(* IEC 61131-3 sources: automationbase/src/OperatingModes, 3 files *)

(* ---- OperatingModes.st ---- *)
NAMESPACE Simatic.Ax.AutomationBase
    /// Operating modes for equipment
    /// Commissioning: Initial setup and testing
    /// Manual: Manual operation with operator control
    /// Automatic: Fully automatic operation with auto-startup
    TYPE
        OperatingModes : (Commissioning, Manual, Automatic) := Manual;
    END_TYPE

END_NAMESPACE

(* ---- IOperatingMode.st ---- *)
NAMESPACE Simatic.Ax.AutomationBase

    {axcode:docs-v0:@simatic-ax/automationbase:OperatingModes.md}
    /// Interface for operating mode providers
    /// Implement this to provide the current operating mode to equipment
    INTERFACE IOperatingMode
        /// Returns the current operating mode (Commissioning, Manual, or Automatic)
        METHOD GetOperatingMode : OperatingModes
        END_METHOD
    END_INTERFACE

END_NAMESPACE

(* ---- OperatingModeManager.st ---- *)
NAMESPACE Simatic.Ax.AutomationBase

    {axcode:docs-v0:@simatic-ax/automationbase:OperatingModes.md}
    /// Generic operating mode manager class
    /// Provides a simple implementation of IOperatingMode with settable mode
    CLASS OperatingModeManager IMPLEMENTS IOperatingMode
        VAR PROTECTED
            /// Current operating mode (default: Manual)
            _currentMode : OperatingModes := OperatingModes#Manual;
        END_VAR

        /// Returns the current operating mode
        METHOD PUBLIC GetOperatingMode : OperatingModes
            GetOperatingMode := _currentMode;
        END_METHOD

        /// Sets the operating mode
        METHOD PUBLIC SetOperatingMode
            VAR_INPUT
                mode : OperatingModes;
            END_VAR
            _currentMode := mode;
        END_METHOD

    END_CLASS

END_NAMESPACE
